Yaskawa INFORM job: AAA.JBI

/JOB
//NAME AAA
//POS
///NPOS 9,0,0,0,0,0
///TOOL 10
///POSTYPE PULSE
///PULSE
C00000=0,-197028,-106872,0,0,0
C00001=1537,-197028,-106872,0,0,0
C00002=-1537,-197028,-106872,0,0,0
C00003=1537,-197028,-106872,0,0,0
C00004=-1537,-197028,-106872,0,0,0
C00005=1537,-197028,-106872,0,0,0
C00006=-1537,-197028,-106872,0,0,0
C00007=1537,-197028,-106872,0,0,0
C00008=-1537,-197028,-106872,0,0,0
//INST
///DATE 2023/03/29 22:56
///ATTR SC,RW
///GROUP1 RB1
NOP
MOVJ C00000 VJ=100.0
MOVJ C00001 VJ=100.0 PL=8
MOVJ C00002 VJ=100.0 PL=8
MOVJ C00003 VJ=100.0 PL=8
MOVJ C00004 VJ=100.0 PL=8
MOVJ C00005 VJ=100.0 PL=8
MOVJ C00006 VJ=100.0 PL=8
MOVJ C00007 VJ=100.0 PL=8
MOVJ C00008 VJ=100.0 PL=8
END
